SYSTEM DistributionStationWithNetwork (* System Configuration *)
  (* Standard: 61499-1 *)
  (* Version 0.3, 2003-12-05, JHC, Rockwell Automation, Renamed from NEWSYSTEM. *)
  APPLICATION APP1
  END_APPLICATION
  DEVICE DEV1 : DeviceType
    RESOURCE Controller : DistributingStation
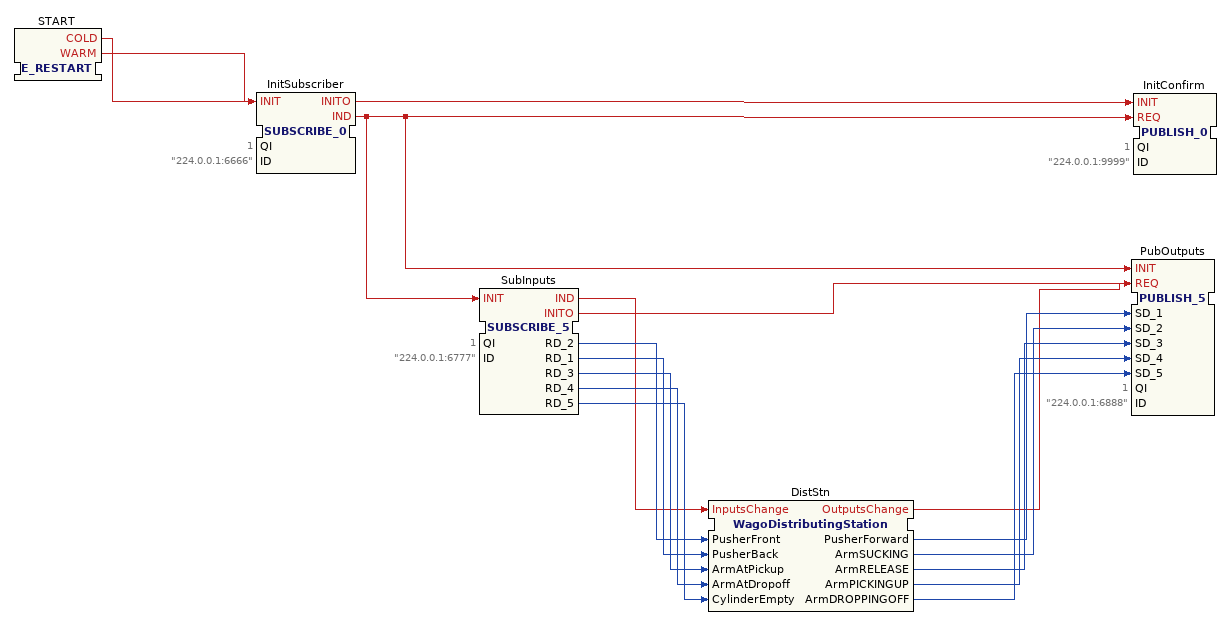
      FBS
        DistStn : WagoDistributingStation;
        SubInputs : SUBSCRIBE_5(QI := 1, ID := "224.0.0.1:6777");
        PubOutputs : PUBLISH_5(QI := 1, ID := "224.0.0.1:6888");
        InitSubscriber : SUBSCRIBE_0(QI := 1, ID := "224.0.0.1:6666");
        START : E_RESTART;
        InitConfirm : PUBLISH_0(QI := 1, ID := "224.0.0.1:9999");
      END_FBS
      EVENT_CONNECTIONS
        START.COLD TO InitSubscriber.INIT;
        InitSubscriber.INITO TO InitConfirm.INIT;
        InitSubscriber.IND TO InitConfirm.REQ;
        START.WARM TO InitSubscriber.INIT;
        InitSubscriber.IND TO SubInputs.INIT;
        InitSubscriber.IND TO PubOutputs.INIT;
        SubInputs.IND TO DistStn.InputsChange;
        SubInputs.INITO TO PubOutputs.REQ;
        DistStn.OutputsChange TO PubOutputs.REQ;
      END_CONNECTIONS
      DATA_CONNECTIONS
        SubInputs.RD_2 TO DistStn.PusherFront;
        SubInputs.RD_1 TO DistStn.PusherBack;
        SubInputs.RD_3 TO DistStn.ArmAtPickup;
        SubInputs.RD_4 TO DistStn.ArmAtDropoff;
        SubInputs.RD_5 TO DistStn.CylinderEmpty;
        DistStn.PusherForward TO PubOutputs.SD_1;
        DistStn.ArmSUCKING TO PubOutputs.SD_2;
        DistStn.ArmRELEASE TO PubOutputs.SD_3;
        DistStn.ArmPICKINGUP TO PubOutputs.SD_4;
        DistStn.ArmDROPPINGOFF TO PubOutputs.SD_5;
      END_CONNECTIONS
    END_RESOURCE
  END_DEVICE
END_SYSTEM
